// TIA Portal V20 export
DATA_BLOCK "DB_WAF"   // DB12
{ S7_Optimized_Access := 'TRUE' }
// stored: MemoryReserve 100
   VAR
      bTest : Array[0..63] of Bool;
      bSpy : Array[0..63] of Bool;
      Sonplas : Struct
         OperateInOutCollision : Bool;
      END_STRUCT;
      BwLoader : Struct
         Safe : Bool;
         Auto : Bool;
      END_STRUCT;
      CtrlInEnable : Bool := true;
      CtrlOutEnable : Bool := true;
      CtrlBwEnable : Bool := true;
      U2States : Byte;
      ResetPartPosition : Bool;
      HMI_Pos : Bool;
      PLC_Pos : Bool;
      NewTag : Bool;
      NewTag_1 : Bool;
   END_VAR
BEGIN
END_DATA_BLOCK
